(* CODESYS project set_in_mode.20190126.1.project

Project tree, tasks and I/O mapping:
  Changsha_Xiangji_ARM_Cortex_A9_xilinx_zynq7000_linux : Changsha Xiangji-ARM Cortex A9(xilinx zynq7000)-linux, Changsha Xiangji Hiden Technology Co.Ltd, version 3.5.10.40
    application Application
      libraries: CAA Types Extern, 3.5.10.0 (CAA Technical Workgroup); VisuDialogs, * (System); CAA Real Time Clock Extern, 3.5.10.0 (CAA Technical Workgroup); CAA Callback Extern, 3.5.11.0 (CAA Technical Workgroup); CAA Can Low Level Extern, 3.5.11.0 (CAA Technical Workgroup); CAA Can Low Level Imp Extern, 3.5.11.0 (CAA Technical Workgroup); SysMem, 3.5.12.0 (System); CAA Net Base Services, 3.5.12.0 (CAA Technical Workgroup); Standard, 3.5.12.0 (System); CAA SerialCom, 3.5.12.0 (CAA Technical Workgroup); CAA File, 3.5.12.0 (CAA Technical Workgroup); CAA DTUtil Extern, 3.5.12.0 (CAA Technical Workgroup); SysFile, 3.5.9.0 (System); SysTypes2 Interfaces, * (System)
      task Task (cyclic, interval 20 ms, priority 10) calls prg_main
      task VISU_TASK (cyclic, interval 100 ms, priority 31) calls VisuElems.Visu_Prg
      parameters/
        data type ST_PARA
        function fn_write_in_mode_file [ST]
        function fn_read_in_mode_file [ST]
      visualisation main
      program prg_main [ST]
      global variables GVL
      funcs/
      text list in_chans
    SoftMotion General Axis Pool
    IoDrvMIC7001 : IoDrvMIC7001, Cyber-MI, version 18.11.1
        output Application.GVL.led_run : BOOL  // LED_run
        unmapped channels: Ai00@C16, Ai01@C28, Ai02@C17, Ai03@C29, Ai04@C30, Ai05@C19, Ai06@C31, Ai07@C20, Ai08@C18, Ai09@D18, Ai10@D20, Ai11@D31, Ai12@D19, Ai13@D30, Ai14@D29, Ai15@D17, Ai16@D28, Ai17@D16, Ai18-Do00@C25, Ai19-Do01@C24, Ai20-Do02@C13, Ai21-Do03@C01, Ai22-Do04@C03, Ai23-Do05@C04, Ai24-Do06@C05, Ai25-Do07@C06, Ai26-Do08@C08, Ai27-Do09@C09, Ai28-Do10@C10, Ai29-Do11@C11, Ai30-Do12@D34, Ai31-Do13@D35, Ai32-Do14@D23, Ai33-Do15@D12, Ai34-Do16@D10, Ai35-Do17@D09, Ai36-Do18@D08, Ai37-Do19@D07, Ai38-Do20@D05, Ai39-Do21@D04,
          Ai40-Do22@D03, Ai41-Do23@D02, Ai42-Do24@C23, Ai43-Do25@C35, Ai44-Do26@D24, Ai45-Do27@D13, Ai46-Ao00@C22, Ai47-Ao01@D14, Ai48_Pi02, Ai49_Out5V, Ai50_VCC, Ai51_VCC_L, Ai52_VCC_R, Ai53_Pwm-i0, Ai54_Pwm-i1, Ai55_Pwm-i2, Ai56_Pwm-i3, Ai57_CPU-T, Ai58_G-x, Ai59_G-y, Ai60_G-z, Ai61-reserved, Ai62-IO-cntr, Ai63-CDS-cntr, Di00-Ai00@C16, Di01-Ai01@C28, Di02-Ai02@C17, Di03-Ai03@C29, Di04-Ai04@C30, Di05-Ai05@C19, Di06-Ai06@C31, Di07-Ai07@C20, Di08-Ai08@C18, Di09-Ai09@D18, Di10-Ai10@D20, Di11-Ai11@D31, Di12-Ai12@D19, Di13-Ai13@D30, Di14-Ai14@D29, Di15-Ai15@D17,
          Di16-Ai16@D28, Di17-Ai17@D16, Di18-Ai18@C25, Di19-Ai19@C24, Di20-Ai20@C13, Di21-Ai21@C01, Di22-Ai22@C03, Di23-Ai23@C04, Di24-Ai24@C05, Di25-Ai25@C06, Di26-Ai26@C08, Di27-Ai27@C09, Di28-Ai28@C10, Di29-Ai29@C11, Di30-Ai30@D34, Di31-Ai31@D35, Di32-Ai32@D23, Di33-Ai33@D12, Di34-Ai34@D10, Di35-Ai35@D09, Di36-Ai36@D08, Di37-Ai37@D07, Di38-Ai38@D05, Di39-Ai39@D04, Di40-Ai40@D03, Di41-Ai41@D02, Di42-Ai42@C23, Di43-Ai43@C35, Di44-Ai44@D24, Di45-Ai45@D13, Di46-Ai46@C22, Di47-Ai47@D14, Di48-Pi00@C15, Di49-Pi01@C14, Di50-Pi02@D22, Di51-Pi03@D21, Di52-reserved, Di53-reserved, Di54-reserved, Di55-reserved,
          Di56-reserved, Di57-reserved, Di58-reserved, Di59-reserved, Di60-reserved, Di61-reserved, Di62-reserved, Di63-reserved, Pi00-Di48@C15, Pi01-Di49@C14, Pi02-Di50@D22, Pi03-Di51@D21, Do00-Ai18@C25, Do01-Ai19@C24, Do02-Ai20@C13, Do03-Ai21@C01, Do04-Ai22@C03, Do05-Ai23@C04, Do06-Ai24@C05, Do07-Ai25@C06, Do08-Ai26@C08, Do09-Ai27@C09, Do10-Ai28@C10, Do11-Ai29@C11, Do12-Ai30@D34, Do13-Ai31@D35, Do14-Ai32@D23, Do15-Ai33@D12, Do16-Ai34@D10, Do17-Ai35@D09, Do18-Ai36@D08, Do19-Ai37@D07, Do20-Ai38@D05, Do21-Ai39@D04, Do22-Ai40@D03, Do23-Ai41@D02, Do24-Ai42@C23, Do25-Ai43@C35, Do26-Ai44@D24, Do27-Ai45@D13,
          Do28-Pwmi00@C33, Do29-Pwmi01@C34, Do30-Pwmi02@D25, Do31-Pwmi03@D26, PWM00@C25, PWM01@C24, PWM02@C13, PWM03@C01, PWM04@C03, PWM05@C04, PWM06@C05, PWM07@C06, PWM08@C08, PWM09@C09, PWM10@C10, PWM11@C11, PWM12@D34, PWM13@D35, PWM14@D23, PWM15@D12, PWM16@D10, PWM17@D09, PWM18@D08, PWM19@D07, PWM20@D05, PWM21@D04, PWM22@D03, PWM23@D02, PWM24@C23, PWM25@C35, PWM26@D24, PWM27@D13, PWM28-Pwmi00@C33, PWM29-Pwmi01@C34, PWM30-Pwmi02@D25, PWM31-Pwmi03@D26, PWM_I_0@C33, PWM_I_1@C34, PWM_I_2@D25, PWM_I_3@D26,
          Ao00-Ai46@C22, Ao01-Ai47@D14, LED_err, LED_usr, ctrl_ai_raw, ctrl_adjust, ctrl_adj0, ctrl_adj1, ctrl_adj2, ctrl_adj3, ctrl_adj4
  5ce3da45-db07-42e7-a21c-a00fff4ed8f6|C:\Users\Administrator\Desktop\robotview1.bmp
  5ce3da45-db07-42e7-a21c-a00fff4ed8f6|C:\Users\Administrator\Desktop\robotview2.bmp
  text list GlobalTextList
  5ce3da45-db07-42e7-a21c-a00fff4ed8f6|C:\Users\Administrator\Desktop\1129.bmp
  5ce3da45-db07-42e7-a21c-a00fff4ed8f6|C:\Users\Administrator\Desktop\robotview0.bmp
*)

// Changsha_Xiangji_ARM_Cortex_A9_xilinx_zynq7000_linux/Application/parameters/ST_PARA
TYPE ST_PARA :
STRUCT
	len:DWORD := 64;   //参数的个数，根据需要设置。设置后最好不变，改变后以前保存的参数作废
	para_val:ARRAY[0..63] OF REAL; 	
	para_ok:BOOL := FALSE;
END_STRUCT
END_TYPE

// Changsha_Xiangji_ARM_Cortex_A9_xilinx_zynq7000_linux/Application/GVL
VAR_GLOBAL
	gRandomNum:DWORD := 146493827;
	led_run:BOOL := FALSE;
END_VAR
VAR_GLOBAL CONSTANT
	inmode_file:STRING:=ANY_TO_STRING("in_mode.txt");
END_VAR

// Changsha_Xiangji_ARM_Cortex_A9_xilinx_zynq7000_linux/Application/prg_main
PROGRAM prg_main  //主控制程序
VAR
	iStat:UINT:= 0;
	tmr_run:ton();
	in_mode:ARRAY[0..47] OF UINT;
	i: INT;
	save_flag :BOOL := FALSE;
	old_index :UINT := 0;
	old_mode :UINT := 0;
	curr_index :UINT:=0;
	curr_mode :UINT := 0;
	changed_flag :BOOL := FALSE;
END_VAR

VAR CONSTANT

END_VAR


CASE iStat OF
	0: //init
		IF fn_read_in_mode_file(ADR(in_mode),48) THEN
			iStat := 20;
			curr_index := 0;
			curr_mode := in_mode[curr_index];
			
			old_index := curr_index;
			old_mode := curr_mode;
		ELSE
			iSTat := 10; //no in_mode file , init with default value
		END_IF
 	10:
		FOR i := 0 TO 47 DO
			in_mode[i] := 0;
		END_FOR
		iStat := 20;
	20:	
		IF save_flag THEN
			iStat := 30;
		END_IF
		
		IF curr_mode <> old_mode THEN
			IF curr_mode <2 OR curr_mode > 3 THEN  
				in_mode[curr_index] := curr_mode;
				old_mode := curr_mode;
				changed_flag := TRUE;
			ELSIF curr_mode = 2 AND curr_index < 8 THEN	
				in_mode[curr_index] := curr_mode;
				old_mode := curr_mode;	
				changed_flag := TRUE;
			ELSIF curr_mode = 2 AND curr_index>9 AND curr_index <18 THEN
				in_mode[curr_index] := curr_mode;
				old_mode := curr_mode;
				changed_flag := TRUE;		
			ELSIF curr_mode = 3 AND (curr_index = 0  OR curr_index = 10) THEN
				in_mode[curr_index] := curr_mode;
				old_mode := curr_mode;
				changed_flag := TRUE;		
			ELSE   //don't support
				curr_mode := old_mode;		
			END_IF
		END_IF
		
		IF curr_index <> old_index THEN
			curr_mode := in_mode[curr_index];
			old_mode := curr_mode;
			old_index := curr_index;
		END_IF
		
	30:
		IF fn_write_in_mode_file(ADR(in_mode), 48) THEN
			save_flag := FALSE;
			iStat := 20;
			changed_flag := FALSE;
		END_IF
END_CASE

tmr_run(in := TRUE, pt := TIME#500MS);
IF tmr_run.Q THEN
	led_run := NOT led_run;
	tmr_run(in := FALSE);
END_IF

END_PROGRAM

// Changsha_Xiangji_ARM_Cortex_A9_xilinx_zynq7000_linux/Application/parameters/fn_read_in_mode_file
FUNCTION fn_read_in_mode_file : BOOL
VAR_INPUT
	pInMode :POINTER TO UINT;
	number:UINT;
END_VAR
VAR
	hFile: RTS_IEC_HANDLE;
	udiOpenError: RTS_IEC_RESULT;
	udiReadError: RTS_IEC_RESULT;
	i :DWORD;
	iTemp: UDINT;
	udiPos: UDINT;
	str: STRING(65535);
	str_size: __XWORD;
	udiByteRead: UDINT;

	len_of_line: INT;
	len_of_number :INT;
	magicNumber:REAL;
	check_sum:REAL:= 0;
	temp_num:REAL;
	index :UINT;
	mode: UINT;
END_VAR

fn_read_in_mode_file := FALSE;

//检测文件是否存在
hFile := sysfileopen(szFile := gvl.inmode_file, am := sysfile.AM_READ, pResult:= ADR(udiOpenError));
IF hFile = RTS_INVALID_HANDLE	THEN  //文件不存在
	RETURN;
END_IF

//文件存在，开始读取内容
udiPos := SysFileSetPos(hFile:=hFile, ulOffset := 0);
udiByteRead := sysfile.SysFileRead(hfile := hFile,pbyBuffer := ADR(str), ulSize := SIZEOF(str), pResult := ADR(udiReadError));
IF udiByteRead < 1 THEN  //读取失败
	sysfile.SysFileClose(hFile := hFile);
	RETURN;
END_IF
sysfile.SysFileClose(hFile);

//读取本行的数字
FOR i := 0 TO number-1 DO
	len_of_number := find(str, WSTRING_TO_STRING("$N"));
	mode := STRING_TO_UINT(left(str,len_of_number-1));
	str := delete(str, len_of_number,1);	
	pInMode[i] := mode;
END_FOR

fn_read_in_mode_file := TRUE;
RETURN;

END_FUNCTION

// Changsha_Xiangji_ARM_Cortex_A9_xilinx_zynq7000_linux/Application/parameters/fn_write_in_mode_file
FUNCTION fn_write_in_mode_file : BOOL
VAR_INPUT
	pInMode :POINTER TO UINT;
	number:UINT;
END_VAR
VAR
	bak_file_prefix:STRING :=ANY_TO_STRING("in_mode_bak_");
	bak_file:STRING := ANY_TO_STRING("");	
	hFile: RTS_IEC_HANDLE;
	udiDeleteError: RTS_IEC_RESULT;
	udiOpenError: RTS_IEC_RESULT;
	udiWriteError: RTS_IEC_RESULT;
	filesize: __XWORD;
	i :DWORD;
	iTemp: UDINT;
	udiPos: UDINT;
	str: STRING(256);
	str_size: __XWORD;
	udiByteWrite: UDINT;
	check_sum:REAL := 0;
	gRandomNum :LWORD := 1;   //系统随机数,每个周期乘以内部传感器的实时值；
END_VAR

fn_write_in_mode_file := FALSE;
gRandomNum := (gRandomNum+1359+ %ID57)*%ID49;

IF number = 0 THEN
	RETURN;
END_IF

//检测文件是否存在，如果存在自动备份
hFile := sysfileopen(szFile := gvl.inmode_file, am := sysfile.AM_READ, pResult:= ADR(udiOpenError));
IF hFile <> RTS_INVALID_HANDLE	THEN  //文件存在
	sysfile.SysFileClose(hFile);  
	bak_file := concat(str1 := bak_file_prefix, str2:= ANY_TO_STRING(gRandomNum));
	filesize := number*16;
	sysfile.SysFileCopy(szDestFileName := bak_file, szSourceFileName := gvl.inmode_file, pulCopied := ADR(filesize));
	sysfile.SysFileDelete(szFileName := gvl.inmode_file);
END_IF

hFile := sysfileopen(szFile := gvl.inmode_file, am := sysfile.AM_WRITE, pResult := ADR(udiOpenError));
IF hFile = RTS_INVALID_HANDLE THEN //创建文件失败
	RETURN;
END_IF
	
udiPos := SysFileSetPos(hFile:=hFile, ulOffset:=0);	
FOR i := 0 TO number-1 DO
	str:= ANY_TO_STRING("");
	str := concat(str, ANY_TO_STRING(pInMode[i]));
	str := concat(str, ANY_TO_STRING("$N"));	
	str_size := ANY_TO_DWORD(len(str));
	udiByteWrite := sysfile.SysFileWrite(hFile := hFile,pbyBuffer := ADR(str),ulSize := str_size, pResult := ADR(udiWriteError));
END_FOR
sysfile.SysFileClose(hFile);
fn_write_in_mode_file := TRUE;

END_FUNCTION

// Changsha_Xiangji_ARM_Cortex_A9_xilinx_zynq7000_linux/Application/main
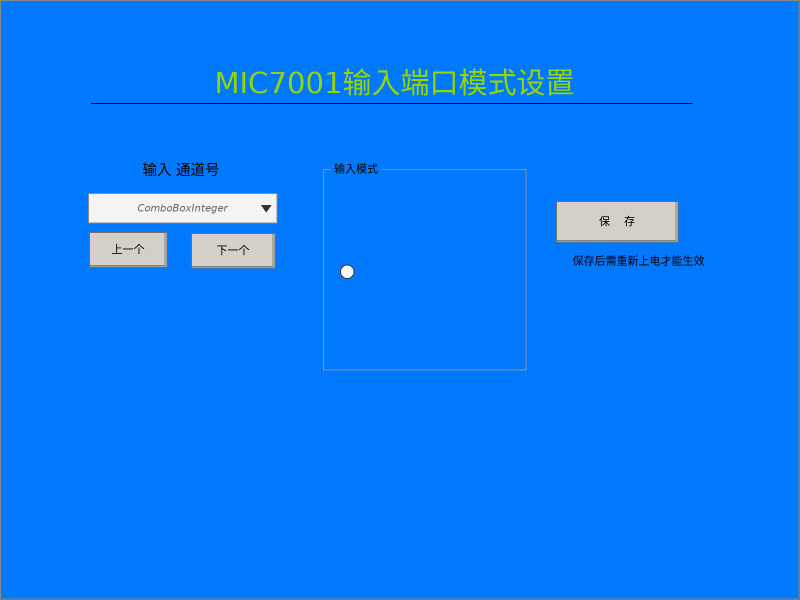
VISUALIZATION main  // 800x600
    ComboBoxInteger (88,193 189x30), variable: prg_main.curr_index, text list: 'in_chans'
    Button (89,232 78x35), "上一个"
        OnMouseClick: execute {
            IF prg_main.curr_index <> 0 THEN
            	prg_main.curr_index := prg_main.curr_index -1;
            ELSE
            	prg_main.curr_index := 47;
            END_IF
        }
    Button (191,233 84x35), "下一个"
        OnMouseClick: execute {
            IF prg_main.curr_index = 47 THEN
            	prg_main.curr_index := 0;
            ELSE
            	prg_main.curr_index := prg_main.curr_index + 1;
            END_IF
        }
    Button (556,201 122x41), "保 存", input disabled if: not prg_main.changed_flag
        OnMouseClick: execute { prg_main.save_flag := true; }
    Label (154,56 481x54), "MIC7001输入端口模式设置"
    Label (91,155 180x30), "输入 通道号"
    Label (553,246 171x30), "保存后需重新上电才能生效"
    Group (323,161 195x209)
        RadioButton (15,17 165x187), variable: prg_main.curr_mode
            Areas[2]: Text=0~36Kohm
            Areas[3]: Text=0~20mA
            Areas[4]: Text=DI_high
            Areas[5]: Text=DI_low
        GroupBox (0,0 203x209), "输入模式"
    Line (23,109)
    Line (91,103) (692,103)
END_VISUALIZATION

(* text list in_chans (id | default)
  0 | AI/DI-00@C16
  1 | AI/DI-01@C28
  2 | AI/DI-02@C17
  3 | AI/DI-03@C29
  4 | AI/DI-04@C30
  5 | AI/DI-05@C19
  6 | AI/DI-06@C31
  7 | AI/DI-07@C20
  8 | AI/DI-08@C18
  9 | AI/DI-09@D18
  10 | AI/DI-10@D20
  11 | AI/DI-11@D31
  12 | AI/DI-12@D19
  13 | AI/DI-13@D30
  14 | AI/DI-14@D29
  15 | AI/DI-15@D17
  16 | AI/DI-16@D28
  17 | AI/DI-17@D16
  18 | AI/DI/DO-18@C25
  19 | AI/DI/DO-19@C24
  20 | AI/DI/DO-20@C13
  21 | AI/DI/DO-21@C01
  22 | AI/DI/DO-22@C03
  23 | AI/DI/DO-23@C04
  24 | AI/DI/DO-24@C05
  25 | AI/DI/DO-25@C06
  26 | AI/DI/DO-26@C08
  27 | AI/DI/DO-27@C09
  28 | AI/DI/DO-28@C10
  29 | AI/DI/DO-29@C11
  30 | AI/DI/DO-30@D34
  31 | AI/DI/DO-31@D35
  32 | AI/DI/DO-32@D23
  33 | AI/DI/DO-33@D12
  34 | AI/DI/DO-34@D10
  35 | AI/DI/DO-35@D09
  36 | AI/DI/DO-36@D08
  37 | AI/DI/DO-37@D07
  38 | AI/DI/DO-38@D05
  39 | AI/DI/DO-39@D04
  40 | AI/DI/DO-40@D03
  41 | AI/DI/DO-41@D02
  42 | AI/DI/PWM-42@C23
  43 | AI/DI/PWM-43@C35
  44 | AI/DI/PWM-44@D24
  45 | AI/DI/PWM-45@D13
  46 | AI/DI/AO-46@C22
  47 | AI/DI/AO-47@D14
   |  *)
